FUNCTION F_Equals : BOOL
VAR_INPUT
    In1 : LREAL;
    In2 : LREAL;
    Delta : LREAL;
END_VAR
VAR
END_VAR

F_Equals := ABS(In1 - In2) < Delta;

END_FUNCTION

(* stored: Version 1.1.0.1, ProductVersion 3.1.4024.3
   POU F_Equals: Id {50cce4b2-d4d9-4bd2-8103-28d757eee48c}, SpecialFunc None *)
